{attribute 'GeneratedUsingTerminal: EL3255-0000-0016'}
{attribute addProperty BoxType "EL3255-0000-0016"}
{attribute addProperty Id "EtcSlaveTerminalBaseRTD_Standard_Channel_1AT %I*RTD_Standard_Channel_A8DF64E310RTD_Standard_Channel_2AT %I*RTD_Standard_Channel_A8DF64E310RTD_Standard_Channel_3AT %I*RTD_Standard_Channel_A8DF64E310RTD_Standard_Channel_4AT %I*RTD_Standard_Channel_A8DF64E310RTD_Standard_Channel_5AT %I*RTD_Standard_Channel_A8DF64E310WcStateAT %I*WcState_9091E0EB2InfoDataAT %I*InfoData_32EB74EA10"}
{attribute addProperty CRC "1594475416"}
{attribute addProperty Size "62"}
TYPE EL3255_5F09C398 EXTENDS EtcSlaveTerminalBase :
STRUCT
	{attribute addProperty Name "RTD_Standard_Channel_1"}
	RTD_Standard_Channel_1 : RTD_Standard_Channel_A8DF64E3;
	{attribute addProperty Name "RTD_Standard_Channel_2"}
	RTD_Standard_Channel_2 : RTD_Standard_Channel_A8DF64E3;
	{attribute addProperty Name "RTD_Standard_Channel_3"}
	RTD_Standard_Channel_3 : RTD_Standard_Channel_A8DF64E3;
	{attribute addProperty Name "RTD_Standard_Channel_4"}
	RTD_Standard_Channel_4 : RTD_Standard_Channel_A8DF64E3;
	{attribute addProperty Name "RTD_Standard_Channel_5"}
	RTD_Standard_Channel_5 : RTD_Standard_Channel_A8DF64E3;
	{attribute addProperty Name "WcState"}
	WcState : WcState_9091E0EB;
	{attribute addProperty Name "InfoData"}
	InfoData : InfoData_32EB74EA;
END_STRUCT
END_TYPE

(* stored: Version 1.2.0.0, ProductVersion 3.1.4024.9
   DUT EL3255_5F09C398: Id {ad5c5f24-9661-4740-8f55-7af51ff6ebb8} *)
